SUBAPPLICATION Ventilsteuerung_Uebung_024 (* Spiegelabfolge (4) *)
  (* Standard: 61499-2 *)
  (* Version 1.0, 2023-10-23, franz *)
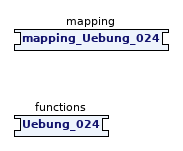
  SUBAPPS
    mapping : mapping_Uebung_024;
    functions : Uebung_024;
  END_SUBAPPS
END_SUBAPPLICATION
